{attribute 'qualified_only'}
{attribute 'strict'}
TYPE E_Drive_JogMode :
(
	eJogMode_0 := 0,//Kontinuierliche Bewegung
	eJogMode_1 		//Tipp Bewegung
);
END_TYPE

(* stored: Version 1.1.0.1
   DUT E_Drive_JogMode: Id {1fd8ca3f-82d8-4f13-80ce-da8e385a7f41} *)
